// SIMATIC S7-200 project (STEP 7-Micro/WIN), CPU 221 REL 01.10

ORGANIZATION_BLOCK MAIN:OB1
TITLE=PROGRAM COMMENTS
BEGIN
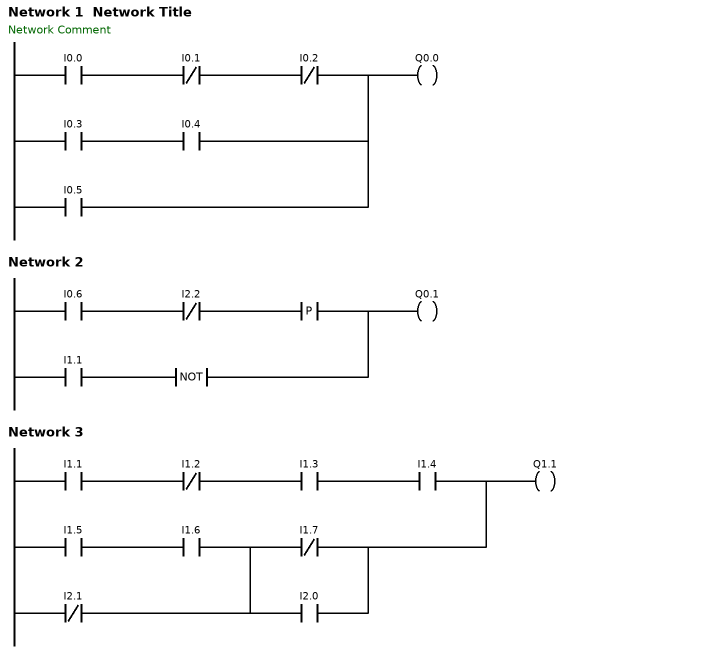
Network 1 // Network Title
// Network Comment
LD     I0.0
AN     I0.1
AN     I0.2
LD     I0.3
A      I0.4
OLD
O      I0.5
=      Q0.0
Network 2
LD     I0.6
AN     I2.2
EU
LD     I1.1
NOT
OLD
=      Q0.1
Network 3
LD     I1.1
AN     I1.2
A      I1.3
A      I1.4
LD     I1.5
A      I1.6
ON     I2.1
LDN    I1.7
O      I2.0
ALD
OLD
=      Q1.1
END_ORGANIZATION_BLOCK
